TYPE ST_ThermalNetworkState :
STRUCT
END_STRUCT
END_TYPE

(* stored: Version 1.1.0.1, ProductVersion 3.1.4024.10
   DUT ST_ThermalNetworkState: Id {cdbdd093-f4bc-4d6a-8042-74c689ffa6d7} *)
